{attribute 'c++_compatible'}
FUNCTION_BLOCK SampleUdpEchoServer IMPLEMENTS ITcIoUdpProtocolRecv
VAR_INPUT
END_VAR
VAR_OUTPUT
END_VAR
VAR
	{attribute 'TcInitSymbol'}
    oid:              OTCID;
	ipUdp:            ITcIoUdpProtocol;
	nUdpPort:         UINT := 10000;
	nReceivedPackets: UINT;
	hrInit:           HRESULT;
	hrSend:           HRESULT;
	
	
	step:          UINT := 0;
	nModes:           UINT := 185;
	nActs:            UINT := 185;

	// row-major, nActs rows x nModes columns: Commands = m2cMatrix * Modes
	m2cMatrix:        ARRAY[0..185*185-1] OF REAL;
	m2cFilename:      STRING := 'C:\TwinCAT\3.1\Boot\eye185.bin';
    fbLoad:           FB_LoadBinaryFile;
	bReload:          BOOL;  // set TRUE (e.g. from a watch window) to reload m2cFilename
	bLoadError:       BOOL;
	nLoadErrId:       UDINT;

	// last received modes and computed commands, kept here so they can be watched/traced
	Modes:            ARRAY[0..185-1] OF REAL;
	Commands:         ARRAY[0..185-1] OF REAL;
	nBadPackets:      UINT;

	counter: UINT := 0;

	value0 AT %Q*:    REAL;
	value1 AT %Q*:    REAL;


	i: INT;
	value: INT;
END_VAR


CASE step OF

0: // default to identity, then try to load the matrix file
	MEMSET(ADR(m2cMatrix), 0, SIZEOF(m2cMatrix));
	FOR i := 0 TO 184 DO
		m2cMatrix[i*185+i] := 1.0;
	END_FOR;
	fbLoad(bExecute := FALSE);
	step := 1;

1: // the load FB must be called every cycle until it is done
    fbLoad(
      sFileName := m2cFilename,
      pDest := ADR(m2cMatrix),
      cbSize := SIZEOF(m2cMatrix),
      bExecute := TRUE
	);
	IF fbLoad.bDone OR fbLoad.bError THEN
		bLoadError := fbLoad.bError;
		nLoadErrId := fbLoad.nErrId;
		fbLoad(bExecute := FALSE);
		step  := 2;
	END_IF

2: // start listening for UDP packets

	IF bReload THEN
		bReload := FALSE;
		step := 0;
	END_IF

	IF ipUdp <> 0 THEN
		ipUdp.CheckReceived();
	END_IF

END_CASE

METHOD FB_exit : BOOL
VAR_INPUT
	bInCopyCode : BOOL; // if TRUE, the exit method is called for exiting an instance that is copied afterwards (online change).
END_VAR
IF (NOT bInCopyCode AND ipUdp <> 0) THEN //Shutdown
     ipUdp.UnregisterReceiver(nUdpPort);
     FW_SafeRelease(ADR(ipUdp));
     FB_exit := TRUE;
ELSE
     FB_exit := FALSE;
END_IF
END_METHOD

METHOD FB_init : BOOL
VAR_INPUT
	bInitRetains : BOOL; // if TRUE, the retain variables are initialized (warm start / cold start)
	bInCopyCode : BOOL;  // if TRUE, the instance afterwards gets moved into the copy code (online change)
END_VAR
IF NOT bInCopyCode THEN // no online change
    IF ipUdp = 0 AND oid <> 0 THEN
     hrInit := FW_ObjMgr_GetObjectInstance(oid:=oid, iid:=TC_GLOBAL_IID_LIST.IID_ITcIoUdpProtocol, pipUnk:=ADR(ipUdp) );
        IF SUCCEEDED(hrInit) THEN 
            IF SUCCEEDED(ipUdp.RegisterReceiver(nUdpPort, THIS^)) THEN //open port
                FB_init := TRUE;
            ELSE 
                FB_init := FALSE; 
                FW_SafeRelease(ADR(ipUdp));
            END_IF
        END_IF
    ELSIF oid = 0 THEN 
        FB_init := FALSE; 
        hrInit := ERR_INVALID_PARAM;                 
    END_IF
END_IF
END_METHOD

METHOD FB_reinit : BOOL
VAR_INPUT
END_VAR
IF (ipUdp <> 0) THEN 
   ipUdp.RegisterReceiver(nUdpPort, THIS^);
   FB_reinit := TRUE;
END_IF
END_METHOD

{attribute 'TcTypeSystem'}
{attribute 'no-analysis'}
{attribute 'c++_compatible'}
{attribute 'minimal_input_size' := '4'}
{attribute 'pack_mode' := '4'}
{warning 'add method implementation '}
METHOD ReceiveData : HRESULT
VAR_INPUT
	ipAddr	: UDINT;
	udpDestPort	: UINT;
	udpSrcPort	: UINT;
	nData	: UDINT;
	pData	: PVOID;
	pVlan	: POINTER TO ETYPE_VLAN_HEADER := 0;
END_VAR

VAR
	dati:  STRING :=  'ciaociao';
	pDati : PVOID :=  0;

END_VAR
nReceivedPackets := nReceivedPackets+1;
//lastReceivedIP.ipadrIPStack := ipAddr;

counter := counter + 1;

pDati := ADR(dati);
IF ipUdp <> 0 THEN

	IF nData >= SIZEOF(Modes) THEN
		// copy first: the UDP payload is not guaranteed to be 4-byte aligned
		MEMCPY(ADR(Modes), pData, SIZEOF(Modes));

		VecMulMatFlat(
			pVec  := ADR(Modes),
			pMat  := ADR(m2cMatrix),
			pRes  := ADR(Commands),
			nVec  := nModes,
			nCols := nActs);

		value0 := Commands[0];
		value1 := Commands[1];

		// send the computed commands back, so the sender can check them
		hrSend := ipUdp.SendData(ipAddr, udpSrcPort, udpDestPort, SIZEOF(Commands), ADR(Commands), TRUE, 0);
	ELSE
		nBadPackets := nBadPackets + 1;
		hrSend := ipUdp.SendData(ipAddr, udpSrcPort, udpDestPort, 8, pDati, TRUE, 0); // send data back
	END_IF
END_IF
END_METHOD

{attribute 'TcTypeSystem'}
{attribute 'no-analysis'}
{attribute 'c++_compatible'}
{attribute 'minimal_input_size' := '4'}
{attribute 'pack_mode' := '4'}
{warning 'add method implementation '}
METHOD TcAddRef : UDINT
END_METHOD

{attribute 'TcTypeSystem'}
{attribute 'no-analysis'}
{attribute 'c++_compatible'}
{attribute 'minimal_input_size' := '4'}
{attribute 'pack_mode' := '4'}
{warning 'add method implementation '}
METHOD TcQueryInterface : HRESULT
VAR_INPUT
	iid	: REFERENCE TO IID;
	pipItf	: POINTER TO PVOID;
END_VAR
VAR
   ipUdpRecv : ITcIoUdpProtocolRecv;
   ipUnknown : ITcUnknown;   
END_VAR
IF GuidsEqual(ADR(iid), ADR(TC_GLOBAL_IID_LIST.IID_ITcIoUdpProtocolRecv)) THEN
    ipUdpRecv := THIS^; // cast to interface pointer
    pipItf^ := ITCUNKNOWN_TO_PVOID(ipUdpRecv);
    TcAddRef();
    TcQueryInterface := S_OK;
ELSIF GuidsEqual(ADR(iid), ADR(TC_GLOBAL_IID_LIST.IID_ITcUnknown)) THEN
    ipUnknown := THIS^; // cast to interface pointer
    pipItf^ := ITCUNKNOWN_TO_PVOID(ipUnknown);
    TcAddRef();
    TcQueryInterface := S_OK;
ELSE
    TcQueryInterface := E_HRESULTAdsErr.NOINTERFACE ; //Call super if this fb extends some other
END_IF
END_METHOD

{attribute 'TcTypeSystem'}
{attribute 'no-analysis'}
{attribute 'c++_compatible'}
{attribute 'minimal_input_size' := '4'}
{attribute 'pack_mode' := '4'}
{warning 'add method implementation '}
METHOD TcRelease : UDINT
END_METHOD

END_FUNCTION_BLOCK

(* stored: Version 1.1.0.1, ProductVersion 3.1.4024.16
   POU SampleUdpEchoServer: Id {9ab8310f-eb11-4595-ad55-314e72a6fce9}, SpecialFunc None
   Method FB_exit: Id {d50239b7-f139-450f-8920-7a3ef99a3ea1}
   Method FB_init: Id {34877cfc-0b22-4fb4-a4e4-fbd786f2bffb}
   Method FB_reinit: Id {d6baa477-95b4-4e81-9ab3-0bc8273c11da}
   Method ReceiveData: Id {3497d4fd-47fe-4e3d-8dcb-1da99f7b9cdf}
   Method TcAddRef: Id {cb5eb8f0-8e85-47c3-9165-4e511c63d67d}
   Method TcQueryInterface: Id {19d31adc-8f1b-4474-83a7-1f1df5e3e5fc}
   Method TcRelease: Id {54c2922f-ec00-4cbc-a530-6f4aa5e9a3f5} *)
